// TwinCAT 3 PLC project PLC
// ProgramVersion: 3.1.4023.0
// libraries:
//   Tc2_Standard, * (Beckhoff Automation GmbH)
//   Tc2_System, * (Beckhoff Automation GmbH)
//   Tc3_Module, * (Beckhoff Automation GmbH)
// project tree:
//   / PlcTask.TcTTO
//   POUs/ FB_Base.TcPOU, FB_Child.TcPOU (not stored), I_Interface2.TcIO, I_Interface.TcIO, MAIN.TcPOU (not stored)
// real-time tasks:
//   TASK PlcTask: cycle T#10ms, priority 20, ADS port 350

CONFIGURATION PLC
    RESOURCE PLC ON TwinCAT3
        TASK PlcTask(INTERVAL := T#10ms, PRIORITY := 20);
        PROGRAM MAIN WITH PlcTask : MAIN;
    END_RESOURCE
END_CONFIGURATION

// ---- POUs/I_Interface2.TcIO
INTERFACE I_Interface2

END_INTERFACE

// ---- POUs/I_Interface.TcIO
INTERFACE I_Interface

END_INTERFACE

// ---- POUs/FB_Base.TcPOU
FUNCTION_BLOCK FB_Base
VAR_INPUT
    Variable1 : INT;
    Variable2   : DINT;
    Variable3   :REAL;
    Sentence : T_MaxString;
    Conditions : ARRAY[1..6] OF BOOL;
END_VAR
VAR_OUTPUT
END_VAR
VAR
END_VAR

END_FUNCTION_BLOCK
